FUNCTION_BLOCK FB_TelescopeSlewingState EXTENDS FB_TelescopeState
VAR_INPUT
	bAutoTrack		: BOOL := FALSE;
END_VAR
VAR_OUTPUT
END_VAR
VAR
END_VAR

// 
// state
//

IF pMachine^.pControl^._Slew() THEN
	IF bAutoTrack THEN
		pMachine^.State := E_TelescopeState.tracking;
	ELSE
		pMachine^.State := E_TelescopeState.idle;
	END_IF
END_IF

//
// commands
// 

IF bPark THEN
	CASE iStage OF
		0:
			IF pMachine^.pControl^._Stop() THEN
				iStage := 1;
			END_IF
		1:
			pMachine^.State := E_TelescopeState.parking;
			bPark := FALSE;
	END_CASE
END_IF

IF bSlew THEN
	bAutoTrack := FALSE;
	pMachine^.State := E_TelescopeState.slewing;	
	bSlew := FALSE;
END_IF

IF bStop THEN
	IF pMachine^.pControl^._Stop() THEN
		pMachine^.State := E_TelescopeState.idle;
		bStop := FALSE;
	END_IF
END_IF

IF bTrack THEN
	CASE iStage OF
		0:
			IF pMachine^.pControl^._Stop() THEN
				iStage := 1;
			END_IF
		1:
			bAutoTrack := TRUE;
			pMachine^.State := E_TelescopeState.slewing;
			bTrack := FALSE;
	END_CASE
END_IF

END_FUNCTION_BLOCK

(* stored: Version 1.1.0.1, ProductVersion 3.1.4024.15
   POU FB_TelescopeSlewingState: Id {edf837d7-00f7-4665-86d4-0431da6cffec}, SpecialFunc None *)
